// TIA Portal V20 export
DATA_BLOCK "Instance_FB_Caroussel_Voltage_Selection_DB"   // DB111
// stored: AutoNumber false, InstanceOfName FB_Caroussel_Voltage_Selection, InstanceOfType FB
"FB_Caroussel_Voltage_Selection"
   // VAR_INPUT
   //    Emergency_Stop_Release : Bool;
   //    Selected_Voltage_220V : Bool;
   //    Selected_Voltage_127V : Bool;
   //    Carousel_Voltage_Selection : SInt;
   // END_VAR
   // VAR_OUTPUT
   //    Voltage_220V_Selected : Bool;
   //    Voltage_127V_Selected : Bool;
   // END_VAR
   // VAR
   //    Delay_Turn_On_220V { S7_SetPoint := 'True'} : TON_TIME;
   //    Delay_Turn_On_127V { S7_SetPoint := 'True'} : TON_TIME;
   // END_VAR
BEGIN
END_DATA_BLOCK
